(* PLC project poST.project, poSTIDE *)
(* stored: creationDateTime 2021-08-31T00:00:00.000000 *)

FUNCTION TRUNC : ANY_INT
  VAR_INPUT
    in : ANY_REAL;
  END_VAR

END_FUNCTION
